(* Logix 5000 project; controller AMP_Servo_Demo 1769-L16ER-BB1B rev 32.15; software revision 32.05 *)
// Applied Motion Products Inc. demo sample program with AOI for Servo drive and Intergrated Servo Motor.

TASK MainTask (continuous, watchdog 500 ms) : MainProgram, Explicit_Messages

MODULES
   Local : 1769-L16ER-BB1B (PointIO 0, rev 32.15)
      AMP_Axis2 : vendor 60 type 43 code 761 (Ethernet 10.10.10.11, rev 3.3, StandardDataDriven RPI 20 ms)   // Applied Motion Products M5 EtherNet/IP Servo Drive
      AMP_Axis1 : vendor 60 type 43 code 601 (Ethernet 10.10.10.10, rev 3.3, StandardDataDriven RPI 12 ms)   // Applied Motion Products MDX+ EtherNet/IP Integrated Servo Motor
      Discrete_IO : Embedded (PointIO 1, rev 32.11, Output RPI 20 ms)
END_MODULES

TYPE AMP_Alarm_Word_Servo :   // Applied Motion Input Assembly - Alarm Word
STRUCT
   Position_Limit : BOOL;
   CCW_Limit : BOOL;
   CW_Limit : BOOL;
   Over_Temperature : BOOL;
   Internal_Error : BOOL;
   Out_of_Range_Voltage : BOOL;
   Over_Current : BOOL;
   Encoder_Disconnected : BOOL;
   USB_Com_Error : BOOL;
   Regen_Failted : BOOL;
   Peak_Current_Foldback : BOOL;
   Abnormal_StartUp : BOOL;
   Safety_Torque_Off : BOOL;
   Velocity_Limit : BOOL;
   Under_Voltage : BOOL;
   Emergenecy_Stop : BOOL;
   Absolute_Position_Lost : BOOL;
   Absolute_Position_Overflow : BOOL;
   Absolute_Postion_MultiTurn_Error : BOOL;
   Abnormal_Motion_Protection : BOOL;
   EthernetIP_Comm_Error : BOOL;
   Homing_Parameter_Error : BOOL;
END_STRUCT
END_TYPE

TYPE AMP_Input_Assembly_Servo_v2 :   // Applied Motion Servo Drive Input Assembly Version 1.0
STRUCT
   Control_Word_Received : DINT;   // Control Word Status equals to Control Words sent in Output Assembly
   OpCode1_Received : DINT;   // OpCode 1 Status equals to OpCode1 sent in Output Assembly
   Control_Mode : DINT;   // Control Mode Status: Position, Torque, Gear
   Status_Code : DINT;   // Status Code
   Alarm_Code : DINT;   // Alarm Code
   Supply_Voltage : DINT;   // Supply Voltage 0.1 V: ex. 242=24.2V
   Applied_Torque : DINT;   // Total Applied Torque %
   Drive_Temperature : DINT;   // Drive Temperature 0.1 deg C: ex. 305=30.5 C
   Encoder_Position : DINT;   // Encoder Position
   Second_Encoder_Position : DINT;   // Absolute Position
   Position_Error : DINT;   // Position Error in Counts
   Actual_Velocity_RPS : DINT;   // Actual Velocity rev/sec*2: ex. 480=2 rev/sec
   Digital_Outputs : DINT;   // Digital Output Status
   Digital_Inputs : DINT;   // Digital Input Status
   Analog_Output1 : DINT;   // 0 = min V, 16383 = max V
   Analog_Output2 : DINT;   // 0 = min V, 16383 = max V
   Analog_Input1 : DINT;   // 0 = min V, 16383 = max V
   Analog_Input2 : DINT;   // 0 = min V, 16383 = max V
   Torque_Limit : DINT;   // Torque Limit Set Point Feedback
   Second_Encoder_Speed : DINT;   // External Encoder Speed Feedback if any
END_STRUCT
END_TYPE

TYPE AMP_Status_Word_Servo :   // Applied Motion Input Assembly Status Word 'SC'
STRUCT
   Enabled : BOOL;   // Motor Enabled (Motor Disabled if this bit = 0)
   Sampling : BOOL;   // Sampling
   Drive_Fault : BOOL;   // Drive Fault (check Alarm Code)
   In_Position : BOOL;   // In Position (motor is in position)
   Moving : BOOL;   // Moving (motor is moving)
   Jogging : BOOL;   // Jogging (currently in jog mode)
   Stopping : BOOL;   // Stopping (in the process of stopping from a stop command)
   Waiting : BOOL;   // Waiting (for an input; executing a WI command)
   Saving : BOOL;   // Saving (parameter data is being saved)
   Alarm_Present : BOOL;   // Alarm present (check Alarm Code)
   Homing : BOOL;   // Homing (executing an SH command)
   Wait_Time : BOOL;   // Waiting (for time; executing a WD or WT command)
   Wizard_Running : BOOL;   // Wizard running (Timing Wizard is running)
   Checking_Encoder : BOOL;   // Checking encoder (Timing Wizard is running)
   Q_Program_Running : BOOL;   // Q Program is running
   Servo_Ready : BOOL;   // Servo Ready;Initializing (happens at power up)
   CSP_Following : BOOL;
   In_Velocity : BOOL;   // Velocity Reached
   Zero_Speed : BOOL;   // Motor is standstill
   Torque_Reached : BOOL;   // Toruqe Target Reached
   In_Torque : BOOL;   // Current Control Mode is Torque
   Group2_PID : BOOL;   // The Second Set of Gain is Valid
   Secondary_Control_Mode : BOOL;   // Second Control Mode is in Operation
   Velocity_Reached : BOOL;   // Velocity Target Reached
   Homing_Complete : BOOL;   // Homing Completed Feedback
END_STRUCT
END_TYPE

ADD_ON_INSTRUCTION AMP_Absolute_Move   (* revision 1.0, vendor Applied Motion Products Inc. *)
// Applied Motion - Motor Absolute Move - AOI
// Help:
// The Absolute Move AOI is used to move an axis to a specified absolute position(FP).
VAR_IN_OUT
   Input : DINT[20]; {required}   // Drive Input Assembly
        [12]   // Digital_Outputs
        [7]   // Drive_Temperature
        [2]   // Control_Mode
        [0]   // Control_Word_Received
        [11]   // Actual_Velocity_RPS
        [4]   // Alarm_Code
        [9]   // Second_Encoder_Position
        [16]   // Analog_Input1
        [10]   // Position_Error
        [17]   // Analog_Input2
        [13]   // Digital_Inputs
        [14]   // Analog_Output1
        [19]   // Second_Encoder_Speed
        [18]   // Torque_Limit
        [3]   // Status_Code
        [15]   // Analog_Output2
        [1]   // OpCode1_Received
        [8]   // Encoder_Position
        [5]   // Supply_Voltage
        [6]   // Applied_Torque
   Output : DINT[11]; {required}   // Drive Output Assembly
        [5]   // Porifle Acceleration
        [6]   // Profile Deceleration
        [0]   // Control Word
        [10]   // Reserved
        [7]   // Target Torque
        [3]   // Target Pos
        [4]   // Target Velocity
        [1]   // OpCode 1
        [2]   // OpCode 2
        [8]   // OpCode 3
        [9]   // OpCode 4
END_VAR
VAR_INPUT
   Start : BOOL; {required}   // Start the Absolute Move
   Position : DINT; {required}   // Destination Position (negative = reverse)
   Speed_rps : REAL; {required}   // Velocity of Move (rev/sec)
   Acc : REAL; {required}   // Acceleration of Move (rev/s/s)
   Dec : REAL; {required}   // Deceleration of Move (rev/s/s)
END_VAR
VAR_OUTPUT
   Sent : BOOL; {access Read Only, visible}   // Move has been sent to drive
   In_Progress : BOOL; {access Read Only, visible}   // Move in progress
   Done : BOOL; {access Read Only, visible}   // Move completed without errors - desired position reached
   Error : BOOL; {access Read Only, visible}   // Move failed to complete - drive not ready or faulted
   State : DINT := 10; {access Read Only}   // Internal state of progress
END_VAR
VAR
   Loc_StatusCode : AMP_Status_Word_Servo; {access None}
   Loc_Input_Assembly : AMP_Input_Assembly_Servo_v2; {access None}
   Loc_Abs_ONS : BOOL;
   Loc_Command_Timeout : TIMER := (PRE := 2000); {access None}   // Timer to output fault if command is not Done
END_VAR

ROUTINE Logic   (* ladder *)
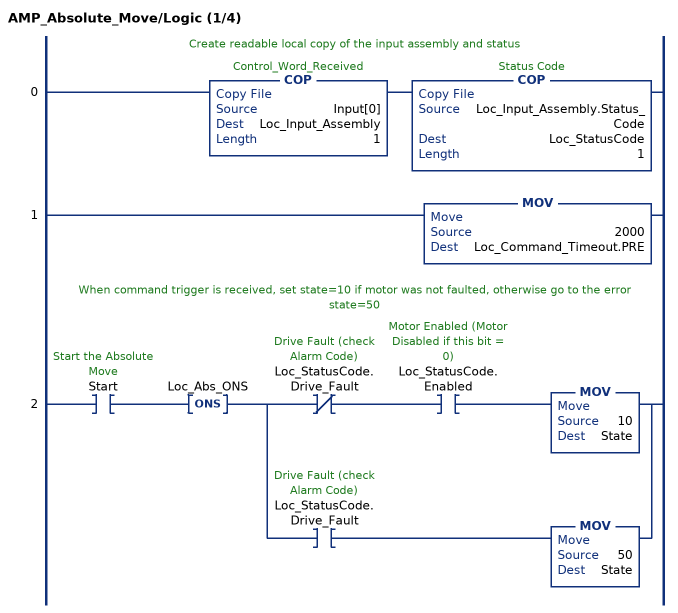
   // Create readable local copy of the input assembly and status
   0: COP(Input[0],Loc_Input_Assembly,1)COP(Loc_Input_Assembly.Status_Code,Loc_StatusCode,1);
   1: MOV(2000,Loc_Command_Timeout.PRE);
   // When command trigger is received, set state=10 if motor was not faulted, otherwise go to the error state=50
   2: XIC(Start)ONS(Loc_Abs_ONS)[XIO(Loc_StatusCode.Drive_Fault) XIC(Loc_StatusCode.Enabled) MOV(10,State) ,XIC(Loc_StatusCode.Drive_Fault) MOV(50,State) ];
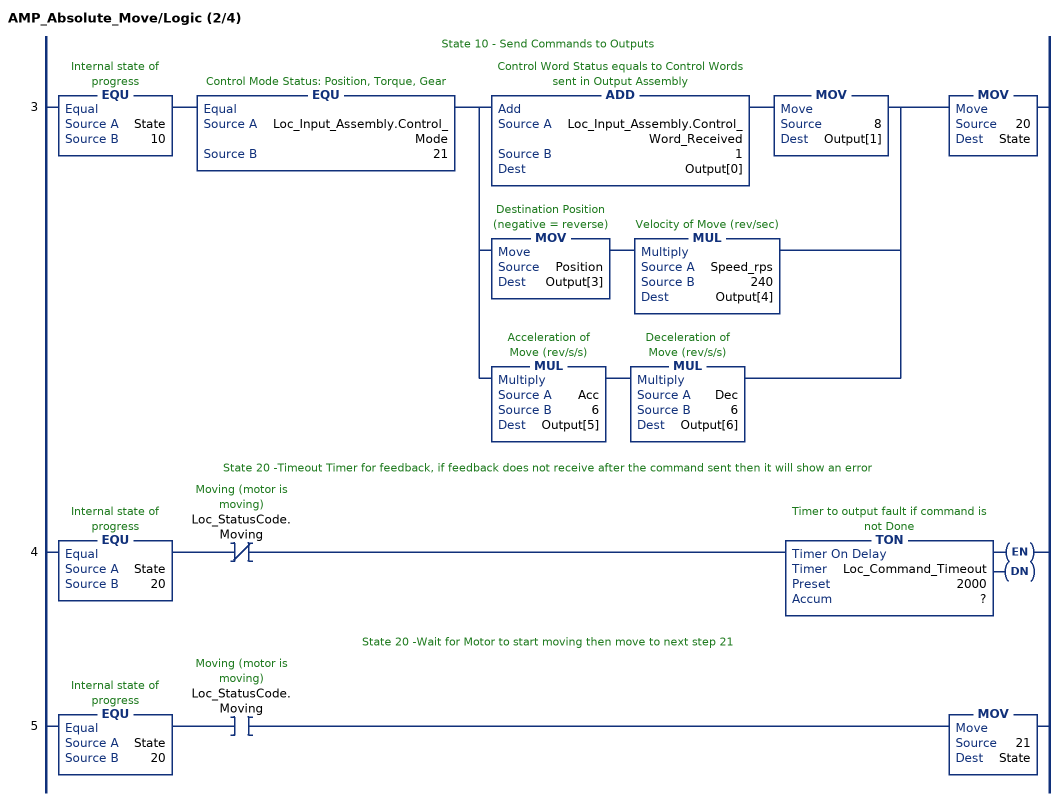
   // State 10 - Send Commands to Outputs
   3: EQU(State,10)EQU(Loc_Input_Assembly.Control_Mode,21)[ADD(Loc_Input_Assembly.Control_Word_Received,1,Output[0]) MOV(8,Output[1]) ,MOV(Position,Output[3]) MUL(Speed_rps,240,Output[4]) ,MUL(Acc,6,Output[5]) MUL(Dec,6,Output[6]) ]MOV(20,State);
   // State 20 -Timeout Timer for feedback, if feedback does not receive after the command sent then it will show an error
   4: EQU(State,20)XIO(Loc_StatusCode.Moving)TON(Loc_Command_Timeout,?,?);
   // State 20 -Wait for Motor to start moving then move to next step 21
   5: EQU(State,20)XIC(Loc_StatusCode.Moving)MOV(21,State);
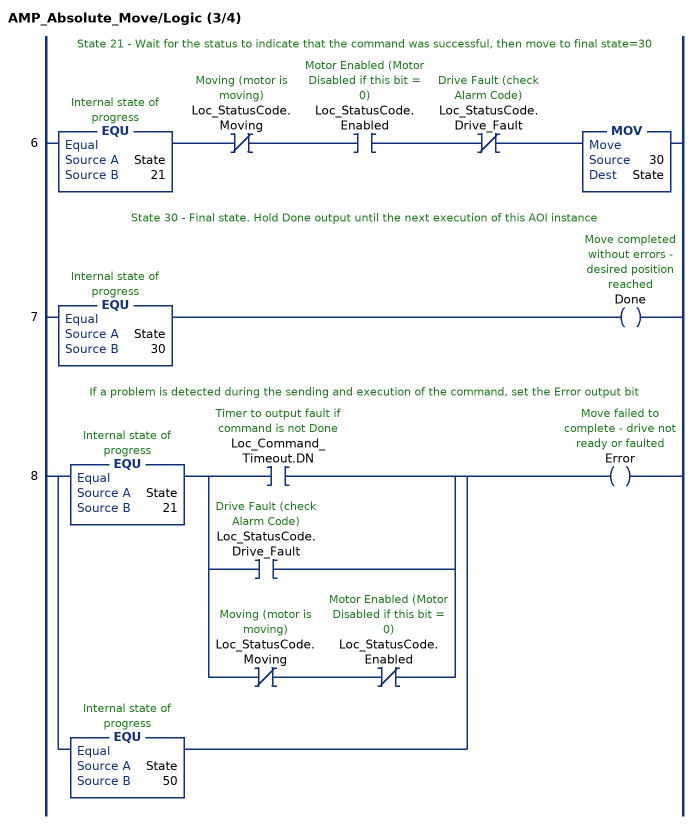
   // State 21 - Wait for the status to indicate that the command was successful, then move to final state=30
   6: EQU(State,21)XIO(Loc_StatusCode.Moving)XIC(Loc_StatusCode.Enabled)XIO(Loc_StatusCode.Drive_Fault)MOV(30,State);
   // State 30 - Final state. Hold Done output until the next execution of this AOI instance
   7: EQU(State,30)OTE(Done);
   // If a problem is detected during the sending and execution of the command, set the Error output bit
   8: [EQU(State,21) [XIC(Loc_Command_Timeout.DN) ,XIC(Loc_StatusCode.Drive_Fault) ,XIO(Loc_StatusCode.Moving) XIO(Loc_StatusCode.Enabled) ] ,EQU(State,50) ]OTE(Error);
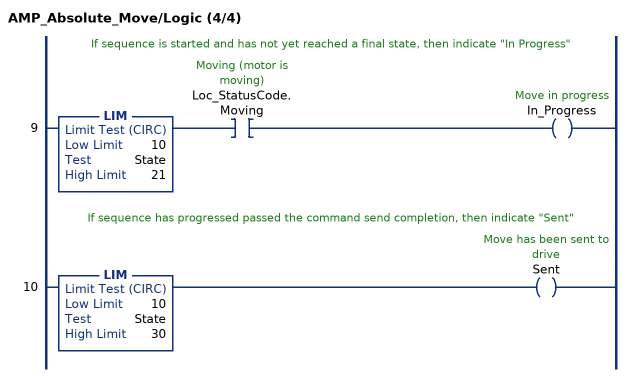
   // If sequence is started and has not yet reached a final state, then indicate "In Progress"
   9: LIM(10,State,21)XIC(Loc_StatusCode.Moving)OTE(In_Progress);
   // If sequence has progressed passed the command send completion, then indicate "Sent"
   10: LIM(10,State,30)OTE(Sent);
END_ROUTINE
END_ADD_ON_INSTRUCTION

ADD_ON_INSTRUCTION AMP_Alarm_Code   (* revision 1.0, vendor Applied Motion Products Inc. *)
// Applied Motion - Alarm Code(AL) AOI
// Help:
// The Alarm Code AOI uses the raw data stored in the Alarm Code word (Element 1 from Input Assembly) to set individual appropriately named boolean outputs.
VAR_INPUT
   Input : DINT; {access Read Only, required}   // Element 5 from Drive Input Assembly
END_VAR
VAR_OUTPUT
   Over_Temp_Fault : BOOL; {access Read Only, visible}   // Over temperature error
   Position_Error_Fault : BOOL; {access Read Only, visible}   // Position Error Limit Fault
   Internal_Error_Fault : BOOL; {access Read Only, visible}   // Internal error fault
   Out_of_Range_Voltage_Fault : BOOL; {access Read Only, visible}   // Power voltage over range
   Over_Current_Fault : BOOL; {access Read Only, visible}   // Over current occured
   Safety_Torque_Off_Fault : BOOL; {access Read Only, visible}   // STO fault occured
   Encoder_Disconnected_Fault : BOOL; {access Read Only, visible}   // Encoder is disconnected
   Velocity_Exceed_Limit_Fault : BOOL; {access Read Only, visible}   // Velocity limit fault
   Abnormal_Motion_Protection_Fault : BOOL; {access Read Only, visible}   // Abnormal motion protection fault
   EthernetIP_Comm_Fault : BOOL; {access Read Only, visible}   // Communication error
   Hybrid_Deviation_Fault : BOOL; {access Read Only, visible}   // Hybrid deviation error fault (full closed loop operationl)
   Secondary_Encoder_Disconnected_Fault : BOOL; {access Read Only, visible}   // Secondary Encoder is not connected (full closed loop operation)
   Emergenecy_Stop_Warning : BOOL; {access Read Only, visible}   // Emergency stop is on
   Regen_Failed_Warning : BOOL; {access Read Only, visible}   // Regen failed warning
   CCW_Limit_Warning : BOOL; {access Read Only, visible}   // Counterclockwise limit
   CW_Limit_Warning : BOOL; {access Read Only, visible}   // Clockwise limit
   Peak_Current_Foldback_Warning : BOOL; {access Read Only, visible}   // Peak Current CP foldback error
   Abnormal_StartUp_Warning : BOOL; {access Read Only, visible}   // Abnormal Start of the motor
   Abnormal_Communication_Warning : BOOL; {access Read Only, visible}   // Abnormal Communication
   Under_Voltage_Warning : BOOL; {access Read Only, visible}   // Undervoltage supply error
   Absolute_Position_Lost_Warning : BOOL; {access Read Only, visible}   // Absolute position lost error
   Absolute_Position_Overflow_Warning : BOOL; {access Read Only, visible}   // Absolute position overflow error
   Absolute_Postion_MultiTurn_Warning : BOOL; {access Read Only, visible}   // Absolute multiturn error
   Homing_Parameter_Warning : BOOL; {access Read Only, visible}   // Wrong homing parameter entered
   Phase_Lost_Warning : BOOL; {access Read Only, visible}   // Motor main power phase lost
   Absolute_Battery_Encoder_Voltage_Warning : BOOL; {access Read Only, visible}   // Absolute Encoder battey is under voltage
   Reserved : INT; {access Read Only}
END_VAR

ROUTINE Logic   (* ladder *)
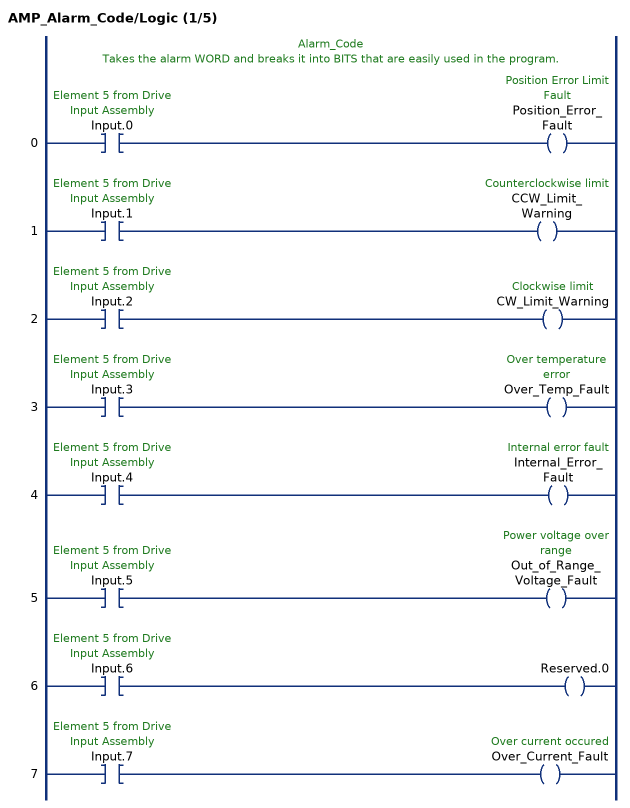
   // Alarm_Code
   // Takes the alarm WORD and breaks it into BITS that are easily used in the program.
   0: XIC(Input.0)OTE(Position_Error_Fault);
   1: XIC(Input.1)OTE(CCW_Limit_Warning);
   2: XIC(Input.2)OTE(CW_Limit_Warning);
   3: XIC(Input.3)OTE(Over_Temp_Fault);
   4: XIC(Input.4)OTE(Internal_Error_Fault);
   5: XIC(Input.5)OTE(Out_of_Range_Voltage_Fault);
   6: XIC(Input.6)OTE(Reserved.0);
   7: XIC(Input.7)OTE(Over_Current_Fault);
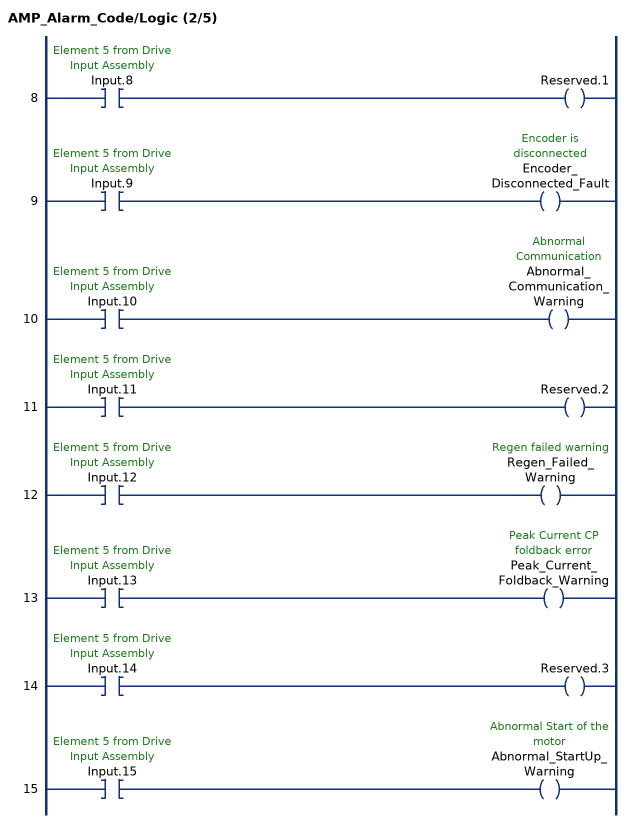
   8: XIC(Input.8)OTE(Reserved.1);
   9: XIC(Input.9)OTE(Encoder_Disconnected_Fault);
   10: XIC(Input.10)OTE(Abnormal_Communication_Warning);
   11: XIC(Input.11)OTE(Reserved.2);
   12: XIC(Input.12)OTE(Regen_Failed_Warning);
   13: XIC(Input.13)OTE(Peak_Current_Foldback_Warning);
   14: XIC(Input.14)OTE(Reserved.3);
   15: XIC(Input.15)OTE(Abnormal_StartUp_Warning);
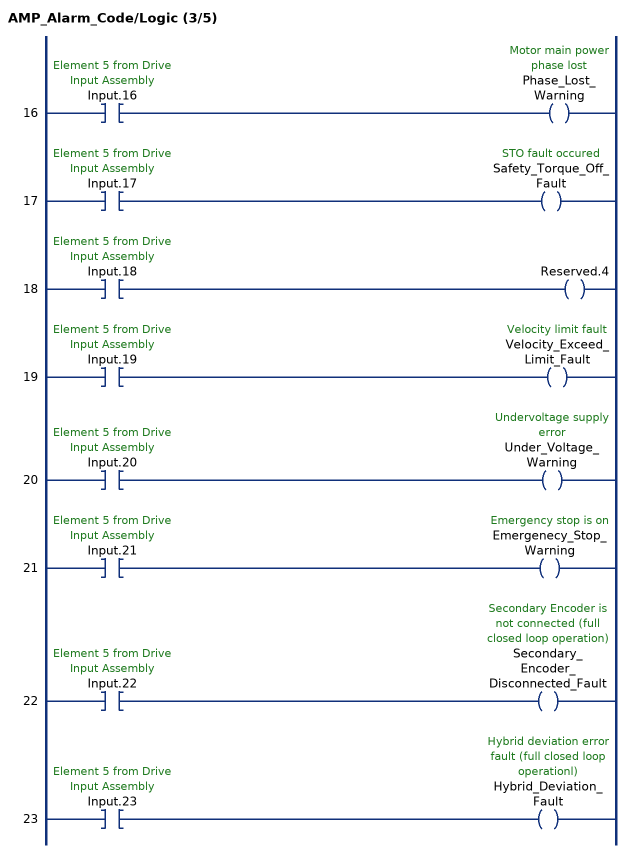
   16: XIC(Input.16)OTE(Phase_Lost_Warning);
   17: XIC(Input.17)OTE(Safety_Torque_Off_Fault);
   18: XIC(Input.18)OTE(Reserved.4);
   19: XIC(Input.19)OTE(Velocity_Exceed_Limit_Fault);
   20: XIC(Input.20)OTE(Under_Voltage_Warning);
   21: XIC(Input.21)OTE(Emergenecy_Stop_Warning);
   22: XIC(Input.22)OTE(Secondary_Encoder_Disconnected_Fault);
   23: XIC(Input.23)OTE(Hybrid_Deviation_Fault);
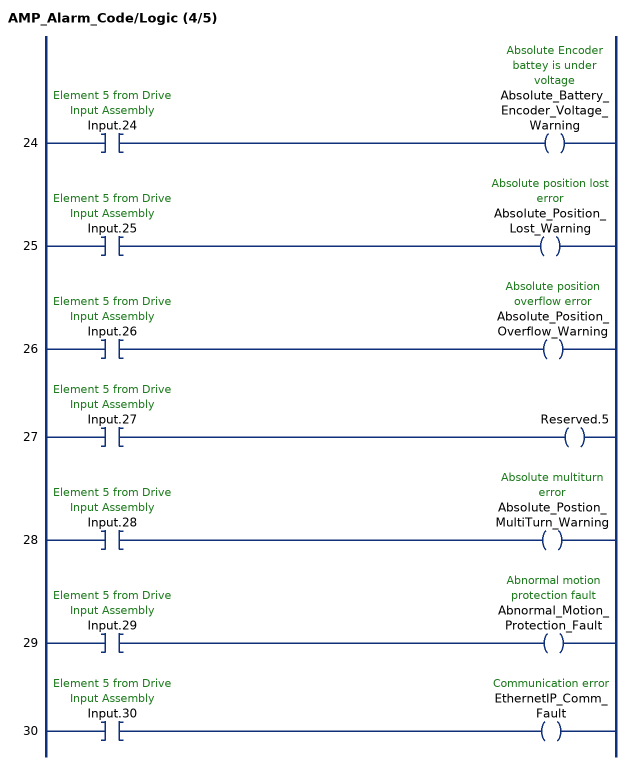
   24: XIC(Input.24)OTE(Absolute_Battery_Encoder_Voltage_Warning);
   25: XIC(Input.25)OTE(Absolute_Position_Lost_Warning);
   26: XIC(Input.26)OTE(Absolute_Position_Overflow_Warning);
   27: XIC(Input.27)OTE(Reserved.5);
   28: XIC(Input.28)OTE(Absolute_Postion_MultiTurn_Warning);
   29: XIC(Input.29)OTE(Abnormal_Motion_Protection_Fault);
   30: XIC(Input.30)OTE(EthernetIP_Comm_Fault);
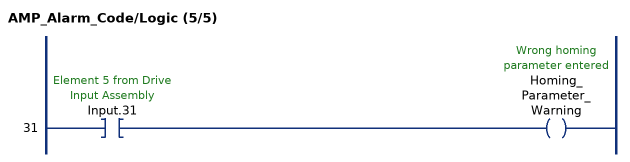
   31: XIC(Input.31)OTE(Homing_Parameter_Warning);
END_ROUTINE
END_ADD_ON_INSTRUCTION

ADD_ON_INSTRUCTION AMP_Alarm_Reset   (* revision 1.0, vendor Applied Motion Products Inc. *)
// Applied Motion - Motor Alarm Reset - AOI
// Help:
// This AOI Reset Active Alarms(AX).
VAR_IN_OUT
   Input : DINT[20]; {required}   // Drive Input Assembly
   Output : DINT[11]; {required}   // Drive Output Assembly
        [5]   // Porifle Acceleration
        [6]   // Profile Deceleration
        [0]   // Control Word
        [10]   // Reserved
        [3]   // Target Pos
        [7]   // Target Torque
        [4]   // Target Velocity
        [1]   // OpCode 1
        [2]   // OpCode 2
        [8]   // OpCode 3
        [9]   // OpCode 4
END_VAR
VAR_INPUT
   Reset : BOOL; {required}   // Reset the Drive (on rising edge)
END_VAR
VAR_OUTPUT
   Sent : BOOL; {access Read Only, visible}   // Reset the Drive has been sent to drive
   In_Progress : BOOL; {access Read Only, visible}   // Reset in progress(not used)
   Done : BOOL; {access Read Only, visible}   // Reset completed without errors
   Error : BOOL; {access Read Only, visible}   // Reset failed
   State : DINT := 10; {access Read Only}   // Internal state of progress
END_VAR
VAR
   Loc_StatusCode : AMP_Status_Word_Servo; {access None}
   Loc_Reset_ONS : BOOL;
   Loc_Input_Assembly : AMP_Input_Assembly_Servo_v2; {access None}
   Loc_Command_Timeout : TIMER := (PRE := 2000); {access None}   // Timer to output fault if command is not Done
END_VAR

ROUTINE Logic   (* ladder *)
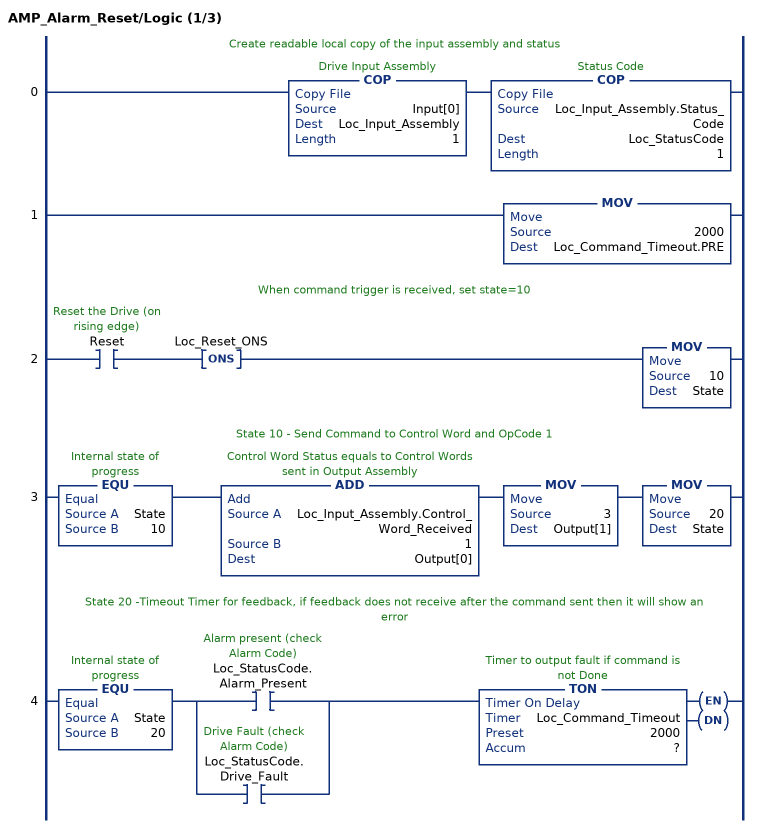
   // Create readable local copy of the input assembly and status
   0: COP(Input[0],Loc_Input_Assembly,1)COP(Loc_Input_Assembly.Status_Code,Loc_StatusCode,1);
   1: MOV(2000,Loc_Command_Timeout.PRE);
   // When command trigger is received, set state=10
   2: XIC(Reset)ONS(Loc_Reset_ONS)MOV(10,State);
   // State 10 - Send Command to Control Word and OpCode 1
   3: EQU(State,10)ADD(Loc_Input_Assembly.Control_Word_Received,1,Output[0])MOV(3,Output[1])MOV(20,State);
   // State 20 -Timeout Timer for feedback, if feedback does not receive after the command sent then it will show an error
   4: EQU(State,20)[XIC(Loc_StatusCode.Alarm_Present) ,XIC(Loc_StatusCode.Drive_Fault) ]TON(Loc_Command_Timeout,?,?);
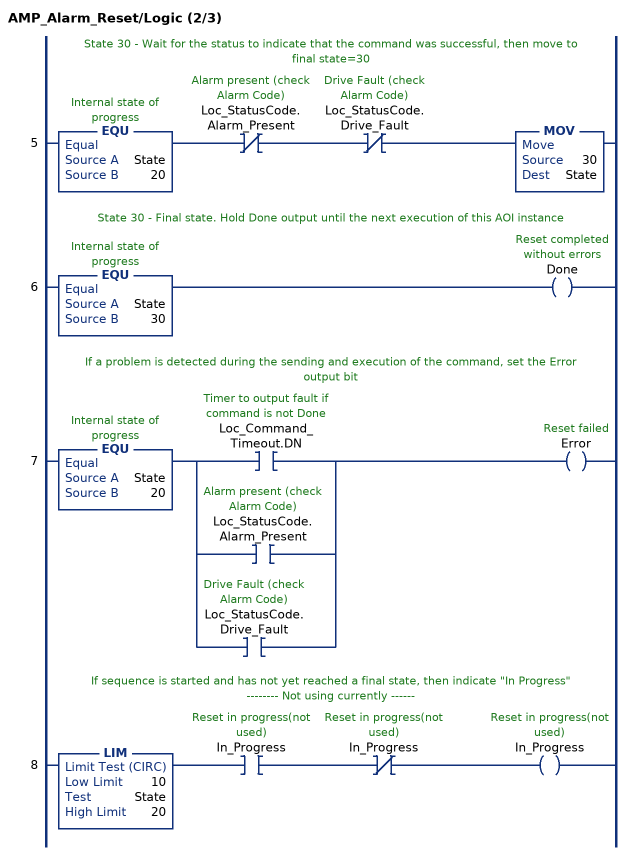
   // State 30 - Wait for the status to indicate that the command was successful, then move to final state=30
   5: EQU(State,20)XIO(Loc_StatusCode.Alarm_Present)XIO(Loc_StatusCode.Drive_Fault)MOV(30,State);
   // State 30 - Final state. Hold Done output until the next execution of this AOI instance
   6: EQU(State,30)OTE(Done);
   // If a problem is detected during the sending and execution of the command, set the Error output bit
   7: EQU(State,20)[XIC(Loc_Command_Timeout.DN) ,XIC(Loc_StatusCode.Alarm_Present) ,XIC(Loc_StatusCode.Drive_Fault) ]OTE(Error);
   // If sequence is started and has not yet reached a final state, then indicate "In Progress"
   // -------- Not using currently ------
   8: LIM(10,State,20)XIC(In_Progress)XIO(In_Progress)OTE(In_Progress);
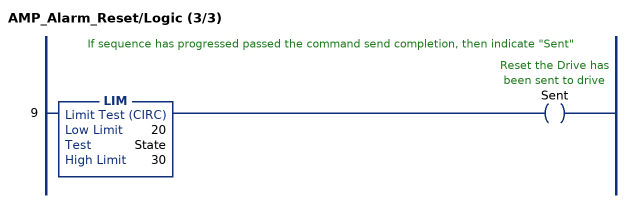
   // If sequence has progressed passed the command send completion, then indicate "Sent"
   9: LIM(20,State,30)OTE(Sent);
END_ROUTINE
END_ADD_ON_INSTRUCTION

ADD_ON_INSTRUCTION AMP_Crash_Stop   (* revision 1.0, vendor Applied Motion Products Inc. *)
// Applied Motion - Stop/Kill using Maximum Deceleration - AOI
// Help:
// This AOI immediately Stop the Motor Jogging/Moving(SK).
VAR_IN_OUT
   Input : DINT[20]; {required}   // Drive Input Assembly
        [12]   // Digital_Outputs
        [7]   // Drive_Temperature
        [2]   // Control_Mode
        [9]   // Second_Encoder_Position
        [0]   // Control_Word_Received
        [11]   // Actual_Velocity_RPS
        [4]   // Alarm_Code
        [19]   // Second_Encoder_Speed
        [16]   // Analog_Input1
        [17]   // Analog_Input2
        [10]   // Position_Error
        [3]   // Status_Code
        [13]   // Digital_Inputs
        [14]   // Analog_Output1
        [15]   // Analog_Output2
        [1]   // OpCode1_Received
        [8]   // Encoder_Position
        [18]   // Torque_Limit
        [5]   // Supply_Voltage
        [6]   // Applied_Torque
   Output : DINT[11]; {required}   // Drive Output Assembly
        [5]   // Porifle Acceleration
        [6]   // Profile Deceleration
        [0]   // Control Word
        [10]   // Reserved
        [7]   // Target Torque
        [3]   // Target Pos
        [4]   // Target Velocity
        [1]   // OpCode 1
        [2]   // OpCode 2
        [8]   // OpCode 3
        [9]   // OpCode 4
END_VAR
VAR_INPUT
   Stop : BOOL; {required}   // Crash Stop the drive axis (on rising edge)
END_VAR
VAR_OUTPUT
   Sent : BOOL; {access Read Only, visible}   // Stop has been sent to drive
   In_Progress : BOOL; {access Read Only, visible}   // Stop in progress
   Done : BOOL; {access Read Only, visible}   // Stop completed without errors - Servo is not moving
   Error : BOOL; {access Read Only, visible}   // Stop failed - drive not stopped or faulted
   State : DINT := 10; {access Read Only}   // Internal state of progress
END_VAR
VAR
   Loc_Stop_ONS : BOOL;
   Loc_StatusCode : AMP_Status_Word_Servo; {access None}
   Loc_Input_Assembly : AMP_Input_Assembly_Servo_v2; {access None}
END_VAR

ROUTINE Logic   (* ladder *)
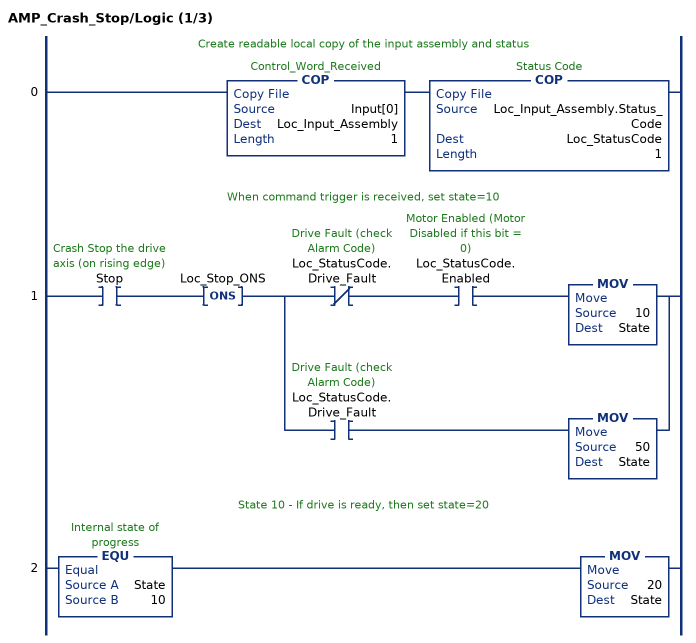
   // Create readable local copy of the input assembly and status
   0: COP(Input[0],Loc_Input_Assembly,1)COP(Loc_Input_Assembly.Status_Code,Loc_StatusCode,1);
   // When command trigger is received, set state=10
   1: XIC(Stop)ONS(Loc_Stop_ONS)[XIO(Loc_StatusCode.Drive_Fault) XIC(Loc_StatusCode.Enabled) MOV(10,State) ,XIC(Loc_StatusCode.Drive_Fault) MOV(50,State) ];
   // State 10 - If drive is ready, then set state=20
   2: EQU(State,10)MOV(20,State);
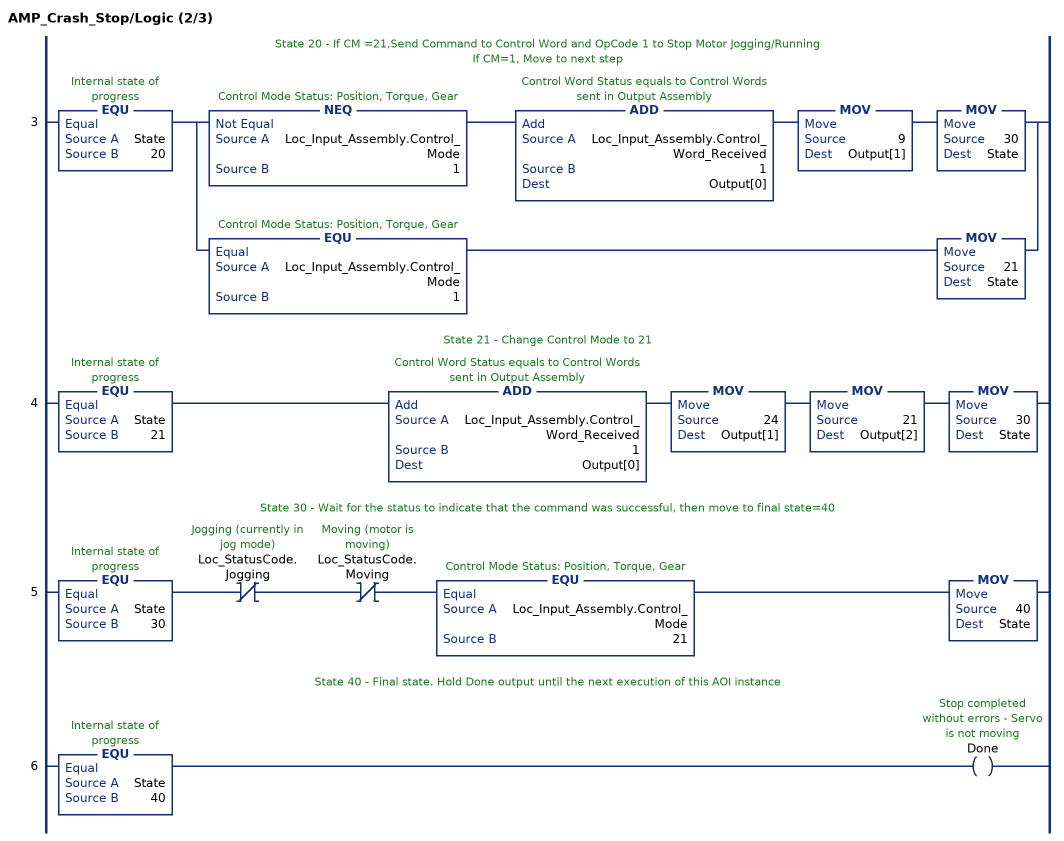
   // State 20 - If CM =21,Send Command to Control Word and OpCode 1 to Stop Motor Jogging/Running
   // If CM=1, Move to next step
   3: EQU(State,20)[NEQ(Loc_Input_Assembly.Control_Mode,1) ADD(Loc_Input_Assembly.Control_Word_Received,1,Output[0]) MOV(9,Output[1]) MOV(30,State) ,EQU(Loc_Input_Assembly.Control_Mode,1) MOV(21,State) ];
   // State 21 - Change Control Mode to 21
   4: EQU(State,21)ADD(Loc_Input_Assembly.Control_Word_Received,1,Output[0])MOV(24,Output[1])MOV(21,Output[2])MOV(30,State);
   // State 30 - Wait for the status to indicate that the command was successful, then move to final state=40
   5: EQU(State,30)XIO(Loc_StatusCode.Jogging)XIO(Loc_StatusCode.Moving)EQU(Loc_Input_Assembly.Control_Mode,21)MOV(40,State);
   // State 40 - Final state. Hold Done output until the next execution of this AOI instance
   6: EQU(State,40)OTE(Done);
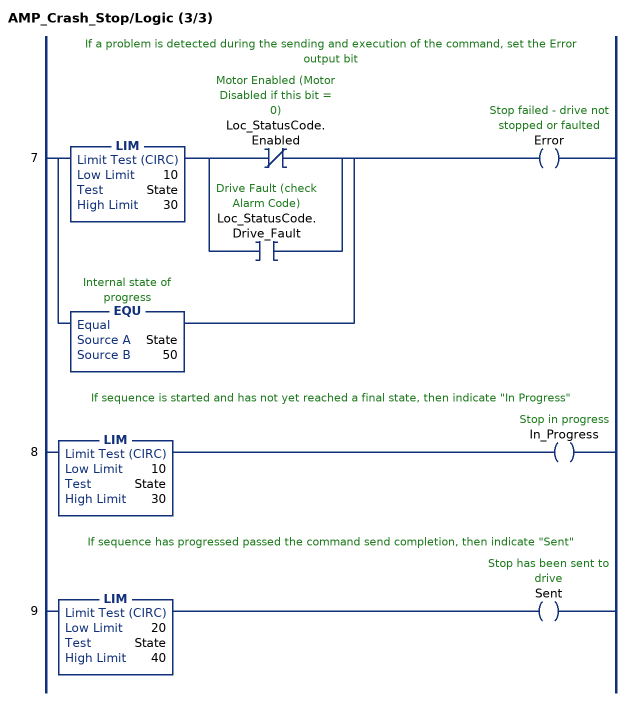
   // If a problem is detected during the sending and execution of the command, set the Error output bit
   7: [LIM(10,State,30) [XIO(Loc_StatusCode.Enabled) ,XIC(Loc_StatusCode.Drive_Fault) ] ,EQU(State,50) ]OTE(Error);
   // If sequence is started and has not yet reached a final state, then indicate "In Progress"
   8: LIM(10,State,30)OTE(In_Progress);
   // If sequence has progressed passed the command send completion, then indicate "Sent"
   9: LIM(20,State,40)OTE(Sent);
END_ROUTINE
END_ADD_ON_INSTRUCTION

ADD_ON_INSTRUCTION AMP_DI_Monitor   (* revision 1.0, vendor Applied Motion Products Inc. *)
// This AOI Monitor available Digital Input Status
// Help:
// Depending on which Drive/Motor Model you have, the number of IO Changes, Ignore extra IO monitoring
// 1 Represent Off/Open, 0 Represent On/Close
VAR_IN_OUT
   Input : DINT[20]; {required}   // Drive Input Assembly
END_VAR
VAR_OUTPUT
   DI_1 : BOOL; {visible}   // Digital Input 1, On = Input Opened, Off = Input Closed
   DI_2 : BOOL; {visible}   // Digital Input 2, On = Input Opened, Off = Input Closed
   DI_3 : BOOL; {visible}   // Digital Input 3, On = Input Opened, Off = Input Closed
   DI_4 : BOOL; {visible}   // Digital Input 4, On = Input Opened, Off = Input Closed
   DI_5 : BOOL; {visible}   // Digital Input 5, On = Input Opened, Off = Input Closed
   DI_6 : BOOL; {visible}   // Digital Input 6, On = Input Opened, Off = Input Closed
   DI_7 : BOOL; {visible}   // Digital Input 7, On = Input Opened, Off = Input Closed
   DI_8 : BOOL; {visible}   // Digital Input 8, On = Input Opened, Off = Input Closed
END_VAR
VAR
   Loc_StatusCode : AMP_Status_Word_Servo; {access None}
   Loc_Input_Assembly : AMP_Input_Assembly_Servo_v2; {access None}
   Inputs_DI : DINT; {access None}
END_VAR

ROUTINE Logic   (* ladder *)
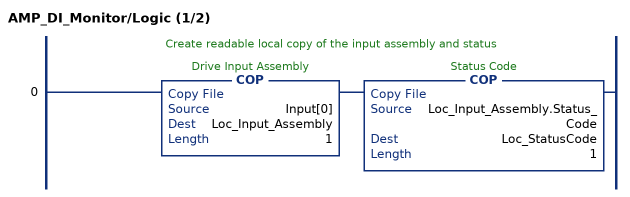
   // Create readable local copy of the input assembly and status
   0: COP(Input[0],Loc_Input_Assembly,1)COP(Loc_Input_Assembly.Status_Code,Loc_StatusCode,1);
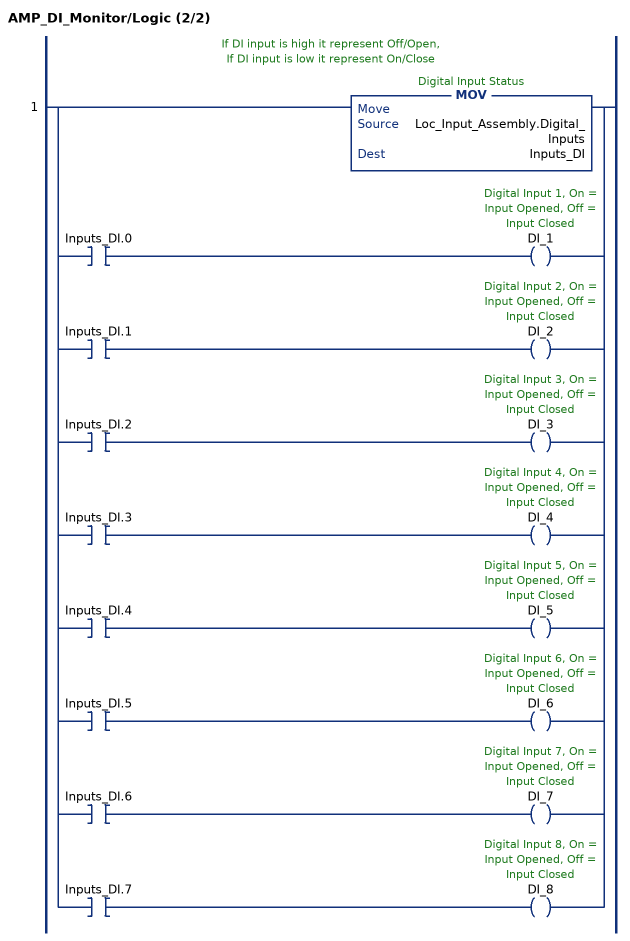
   // If DI input is high it represent Off/Open,
   // If DI input is low it represent On/Close
   1: [MOV(Loc_Input_Assembly.Digital_Inputs,Inputs_DI) ,XIC(Inputs_DI.0) OTE(DI_1) ,XIC(Inputs_DI.1) OTE(DI_2) ,XIC(Inputs_DI.2) OTE(DI_3) ,XIC(Inputs_DI.3) OTE(DI_4) ,XIC(Inputs_DI.4) OTE(DI_5) ,XIC(Inputs_DI.5) OTE(DI_6) ,XIC(Inputs_DI.6) OTE(DI_7) ,XIC(Inputs_DI.7) OTE(DI_8) ];
END_ROUTINE
END_ADD_ON_INSTRUCTION

ADD_ON_INSTRUCTION AMP_DO_Control   (* revision 1.0, vendor Applied Motion Products Inc. *)
// Applied Motion - General Purpose Digital Output Control - AOI
// Help:
// This AOI only Controls Output that are defined as General Purpose Output.
// Depending on which Drive/Motor Model you have, the number of Output Changes, Ignore extra Output.
// Define output number 1-6 and Condition L to Close the output, H to Open the Output.
// As an example, 2L will set output number 2 Close.
// This AOI can be used when Motor is Enable or Disable.
VAR_IN_OUT
   Input : DINT[20]; {required}   // Drive Input Assembly
        [12]   // Digital_Outputs
        [7]   // Drive_Temperature
        [2]   // Control_Mode
        [9]   // Second_Encoder_Position
        [16]   // Analog_Input1
        [4]   // Alarm_Code
        [3]   // Status_Code
        [17]   // Analog_Input2
        [0]   // Control_Word_Received
        [11]   // Actual_Velocity_RPS
        [10]   // Position_Error
        [13]   // Digital_Inputs
        [19]   // Second_Encoder_Speed
        [14]   // Analog_Output1
        [15]   // Analog_Output2
        [1]   // OpCode1_Received
        [18]   // Torque_Limit
        [8]   // Encoder_Position
        [5]   // Supply_Voltage
        [6]   // Applied_Torque
   Output : DINT[11]; {required}   // Drive Output Assembly
        [5]   // Porifle Acceleration
        [6]   // Profile Deceleration
        [0]   // Control Word
        [7]   // Target Torque
        [10]   // Reserved
        [4]   // Target Velocity
        [3]   // Target Pos
        [1]   // OpCode 1
        [2]   // OpCode 2
        [8]   // OpCode 3
        [9]   // OpCode 4
END_VAR
VAR_INPUT
   Execute : BOOL; {required}   // Execute the SCL command 'SO'
   Output_Number : INT; {required}   // Output Number, 1-6
   Condition : SINT; {required}   // Output Condition: H for Open and L for Close Output
END_VAR
VAR_OUTPUT
   DO_1 : BOOL; {visible}   // Digital Output 1, On = Output Closed, Off = Output Opened
   DO_2 : BOOL; {visible}   // Digital Output 2, On = Output Closed, Off = Output Opened
   DO_3 : BOOL; {visible}   // Digital Output 3, On = Output Closed, Off = Output Opened
   DO_4 : BOOL; {visible}   // Digital Output 4, On = Output Closed, Off = Output Opened
   DO_5 : BOOL; {visible}   // Digital Output 5, On = Output Closed, Off = Output Opened
   DO_6 : BOOL; {visible}   // Digital Output 6, On = Output Closed, Off = Output Opened
END_VAR
VAR
   Loc_StatusCode : AMP_Status_Word_Servo;
   Loc_Input_Assembly : AMP_Input_Assembly_Servo_v2;
   Loc_SCL_ONS : BOOL;
   Loc_Outputs_DO : INT; {access None}
   Loc_IO_Condition_Encoded : DINT; {access None}
   Loc_IO1_Number_Encoded : DINT; {access None}
   Loc_State : DINT := 10; {access Read Only}   // Internal state of progress
   Loc_Error : BOOL; {access Read Only}   // Command failed
   Loc_Done : BOOL; {access Read Only}   // Command completed without errors - Drive is Homed
   Loc_In_Progress : BOOL; {access Read Only}   // Command in progress
   Loc_Sent : BOOL; {access Read Only}   // Command has sent
END_VAR

ROUTINE Logic   (* ladder *)
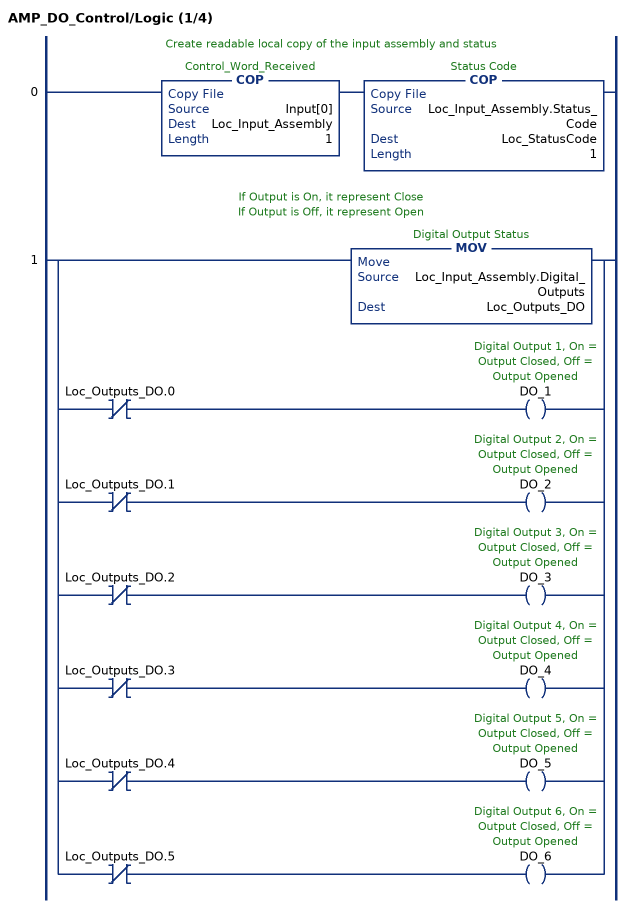
   // Create readable local copy of the input assembly and status
   0: COP(Input[0],Loc_Input_Assembly,1)COP(Loc_Input_Assembly.Status_Code,Loc_StatusCode,1);
   // If Output is On, it represent Close
   // If Output is Off, it represent Open
   1: [MOV(Loc_Input_Assembly.Digital_Outputs,Loc_Outputs_DO) ,XIO(Loc_Outputs_DO.0) OTE(DO_1) ,XIO(Loc_Outputs_DO.1) OTE(DO_2) ,XIO(Loc_Outputs_DO.2) OTE(DO_3) ,XIO(Loc_Outputs_DO.3) OTE(DO_4) ,XIO(Loc_Outputs_DO.4) OTE(DO_5) ,XIO(Loc_Outputs_DO.5) OTE(DO_6) ];
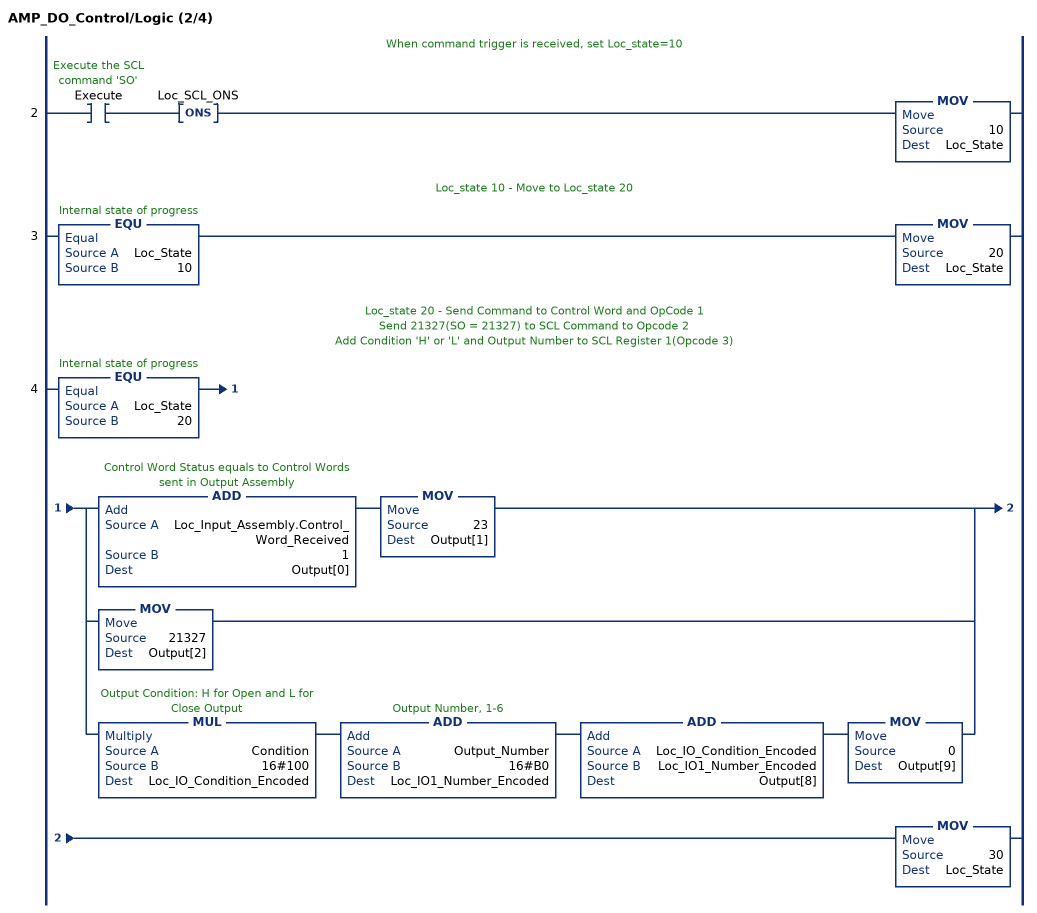
   // When command trigger is received, set Loc_state=10
   2: XIC(Execute)ONS(Loc_SCL_ONS)MOV(10,Loc_State);
   // Loc_state 10 - Move to Loc_state 20
   3: EQU(Loc_State,10)MOV(20,Loc_State);
   // Loc_state 20 - Send Command to Control Word and OpCode 1
   // Send 21327(SO = 21327) to SCL Command to Opcode 2
   // Add Condition 'H' or 'L' and Output Number to SCL Register 1(Opcode 3)
   4: EQU(Loc_State,20)[ADD(Loc_Input_Assembly.Control_Word_Received,1,Output[0]) MOV(23,Output[1]) ,MOV(21327,Output[2]) ,MUL(Condition,16#100,Loc_IO_Condition_Encoded) ADD(Output_Number,16#B0,Loc_IO1_Number_Encoded) ADD(Loc_IO_Condition_Encoded,Loc_IO1_Number_Encoded,Output[8]) MOV(0,Output[9]) ]MOV(30,Loc_State);
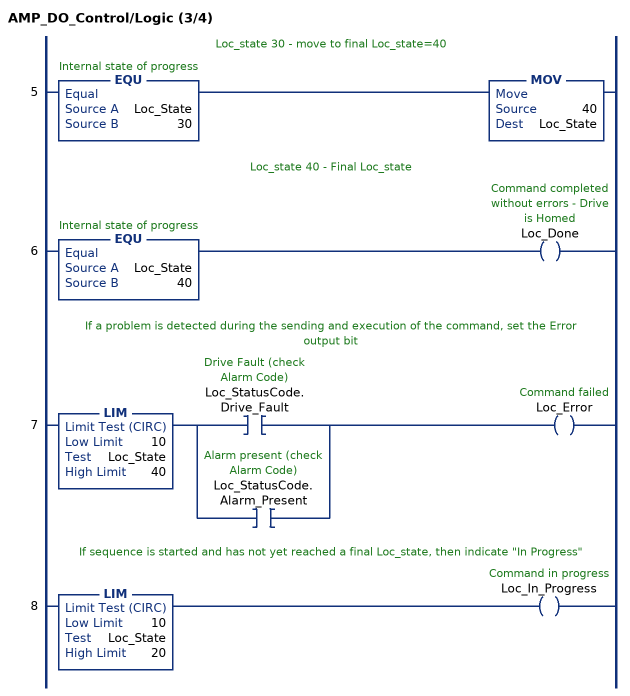
   // Loc_state 30 - move to final Loc_state=40
   5: EQU(Loc_State,30)MOV(40,Loc_State);
   // Loc_state 40 - Final Loc_state
   6: EQU(Loc_State,40)OTE(Loc_Done);
   // If a problem is detected during the sending and execution of the command, set the Error output bit
   7: LIM(10,Loc_State,40)[XIC(Loc_StatusCode.Drive_Fault) ,XIC(Loc_StatusCode.Alarm_Present) ]OTE(Loc_Error);
   // If sequence is started and has not yet reached a final Loc_state, then indicate "In Progress"
   8: LIM(10,Loc_State,20)OTE(Loc_In_Progress);
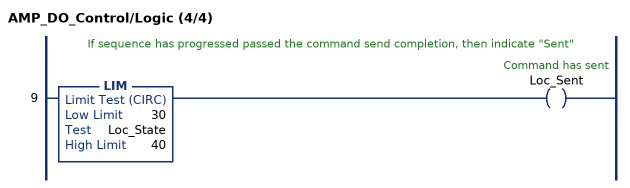
   // If sequence has progressed passed the command send completion, then indicate "Sent"
   9: LIM(30,Loc_State,40)OTE(Loc_Sent);
END_ROUTINE
END_ADD_ON_INSTRUCTION
